FUNCTION_BLOCK FB_BMS_IO

VAR_INPUT
	b_BMSEnable			 AT %Q* : BOOL;
END_VAR

END_FUNCTION_BLOCK

(* stored: Version 1.1.0.1, ProductVersion 3.1.4026.18
   POU FB_BMS_IO: Id {9376410e-3d1b-473f-a7e6-b4fb191e9a9e}, SpecialFunc None *)
